(*
SPDX-FileCopyrightText: © 2026 Oleksandr Tiutyk <trofimich@gmail.com>
SPDX-License-Identifier: MIT
License: https://opensource.org/license/mit
*)

(*!
<summary>Creates a filesystem directory through cyclic task execution.</summary>
<description>
Configure DirectoryPath, PathType, AmsNetId and Timeout before Start and keep them unchanged until STOPPED.
The path must be nonblank and pass PathHelper's limited lexical filter; native services determine whether the
requested operation is supported. This task does not perform an existence precheck or suppress native errors.
Invalid configuration and native errors use the base Task failure and cleanup path. Cancellation waits for
submitted I/O without rolling back completed filesystem changes. Reset clears the native request state and
preserves configuration. Use one owner task per instance.
</description>
*)

{attribute 'no_explicit_call' := 'do not call this function block directly'}
FUNCTION_BLOCK CreateDirectory EXTENDS TOF_Tasks.Task IMPLEMENTS IFileSystemTask
VAR_STAT
	//! <summary>Static type metadata available before the base task initializes its default name.</summary>
	{attribute 'hide'}
	_ClassName : STRING := __POUNAME();
END_VAR
VAR
    _CreateDirectory : Tc2_System.FB_CreateDir;
END_VAR

(*!
<summary>Selects the ADS target for the native filesystem operation.</summary>
<description>
Configure before Start and keep unchanged until STOPPED; the setter stores configuration without submitting
I/O.
</description>
*)
{attribute 'monitoring' := 'call'}
PROPERTY AmsNetId : Tc2_System.T_AmsNetID
GET
AmsNetId := _CreateDirectory.sNetId;
END_GET
SET
_CreateDirectory.sNetId := AmsNetId;
END_SET
END_PROPERTY

(*!
<summary>Provides the concrete type name used in diagnostics.</summary>
<description>
Returns borrowed read-only metadata; keep the instance alive and do not modify the referenced string.
Initialized static storage is ready during base Task.FB_init; this getter has no side effects or exceptions.
</description>
*)
{attribute 'monitoring' := 'call'}
PROPERTY ClassName : REFERENCE TO STRING
GET
ClassName REF= _ClassName;
END_GET
END_PROPERTY

{attribute 'monitoring' := 'call'}
(*!
<summary>Provides the copied path for the next directory operation.</summary>
<description>
Set before Start and keep unchanged until STOPPED. Checked by PathHelper before submission, then interpreted
by the native service using PathType. Assignment does not perform I/O; Reset preserves it.
</description>
*)
PROPERTY DirectoryPath : Tc2_System.T_MaxString
GET
DirectoryPath := _CreateDirectory.sPathName;
END_GET
SET
_CreateDirectory.sPathName := DirectoryPath;
END_SET
END_PROPERTY

(*!
<summary>Provides the library namespace used in diagnostics.</summary>
<description>Returns borrowed read-only namespace storage; do not modify the referenced string.</description>
*)
{attribute 'monitoring' := 'call'}
PROPERTY NamespaceName : REFERENCE TO STRING
GET
NamespaceName REF= CurrentNamespace.Name;
END_GET
END_PROPERTY

(*!
<summary>Resets the native request edge after the task has stopped.</summary>
<description>
Preserves configured inputs and does not undo completed filesystem effects. Pending I/O must finish during
stopping before this hook runs.
</description>
*)
METHOD PROTECTED OnReset
_CreateDirectory(bExecute := FALSE);
END_METHOD

(*!
<summary>Validates the configured path and advances the native directory-create request.</summary>
<description>
Computed diagnostic strings are held in local buffers for the duration of the receiving call without dynamic
string-builder allocations.
</description>
*)
METHOD PROTECTED OnRunning
VAR_OUTPUT
	processingState : TOF_Tasks.TASK_PROCESSING_STATE;
END_VAR
VAR_IN_OUT
	stopReasonMessage : TOF_Core.ERROR_MESSAGE;
END_VAR
VAR	
	pathErrorMessage : WSTRING(255);
	formattedExceptionMessage : TOF_Core.ERROR_MESSAGE;
END_VAR
IF NOT _CreateDirectory.bExecute THEN 
	IF TOF_Core.Strings.IsNullOrWhiteSpace(stringToCheck := _CreateDirectory.sPathName) THEN
		TOF_Core.Exceptions.ThrowDataMemberNotSpecified(
			sourceNamespaceName := NamespaceName,
			sourceClassName := ClassName,
			sourcePOUName := __POUNAME(),
			sourcePosition := __POSITION(),
			dataMemberName := 'DirectoryPath'
		);		
	END_IF
	
	IF NOT PathHelper.IsValidDirectoryPath(directoryPath := _CreateDirectory.sPathName, errorMessage => pathErrorMessage) THEN
		FileSystemExceptions.ThrowInvalidPath(
			sourceNamespaceName := NamespaceName,
			sourceClassName := ClassName,
			sourcePOUName := __POUNAME(),
			sourcePosition := __POSITION(),
			path := _CreateDirectory.sPathName,
			errorMessage := pathErrorMessage
		);
	END_IF
END_IF

_CreateDirectory(bExecute := TRUE);

IF _CreateDirectory.bError THEN
	TOF_Core.WideStrings.Append255(
		formattedExceptionMessage,
		"Error while creating directory '",
		TO_WSTRING(_CreateDirectory.sPathName),
		"'");

	FileSystemExceptions.ThrowFileSystem(
		sourceNamespaceName := NamespaceName,
		sourceClassName := ClassName,
		sourcePOUName := __POUNAME(),
		sourcePosition := __POSITION(),
		message := formattedExceptionMessage,
		errorCode := _CreateDirectory.nErrId
	);
ELSIF NOT _CreateDirectory.bBusy THEN
	processingState := TOF_Tasks.TASK_PROCESSING_STATE.DONE;
END_IF
END_METHOD

(*!
<summary>Waits for an already submitted operation before task termination.</summary>
<description>
Runs for every stop reason. Advances the pending FB with bExecute=FALSE without issuing another request.
Completion does not roll back side effects. Keep configuration and borrowed buffers valid until STOPPED.
</description>
<param name="readyToRelease">TRUE when the underlying FB is no longer busy.</param>
*)
METHOD PROTECTED OnStopping
VAR_OUTPUT
	readyToRelease : BOOL;
END_VAR
IF _CreateDirectory.bBusy THEN
	_CreateDirectory(bExecute := FALSE);
END_IF

readyToRelease := NOT _CreateDirectory.bBusy;
END_METHOD

(*!
<summary>Selects the native path context for the filesystem request.</summary>
<description>
Configure before Start and keep unchanged until STOPPED. It is passed to the native operation, not used as a
path-validity result. Reset preserves it.
</description>
*)
{attribute 'monitoring' := 'call'}
PROPERTY PathType : Tc2_System.E_OpenPath
GET
PathType := _CreateDirectory.ePath;
END_GET
SET
_CreateDirectory.ePath := PathType;
END_SET
END_PROPERTY

(*!
<summary>Reports the size of this concrete instance in bytes.</summary>
*)
{attribute 'monitoring' := 'call'}
PROPERTY SelfSize : ULINT
GET
SelfSize := XSIZEOF(THIS^);
END_GET
END_PROPERTY

(*!
<summary>Configures the timeout passed to native operation requests.</summary>
<description>
Set before Start and keep unchanged until STOPPED. Reset preserves this value. It is not an overall task
deadline or a guarantee of resource release after a timeout.
</description>
*)
{attribute 'monitoring' := 'call'}
PROPERTY Timeout : TIME
GET
Timeout := _CreateDirectory.tTimeout;
END_GET
SET
_CreateDirectory.tTimeout := Timeout;
END_SET
END_PROPERTY

END_FUNCTION_BLOCK

(* stored: Version 1.1.0.1
   POU CreateDirectory: Id {7b0b8920-cd1b-44d1-9ca2-1004e427656c}, SpecialFunc None
   Folder Inputs: Id {cd46d3f1-05ad-4d2a-bb18-250033ee445c}
   Folder Members to override: Id {740079d8-792c-4051-b807-b10023f9c7a1}
   Property AmsNetId: Id {ed338df4-10dc-451a-b64d-a000a295e7f0}
   Get Get: Id {94b5c541-fb9b-4788-a387-16d6d7a06a3f}
   Set Set: Id {477e135b-e114-4f7b-ae5e-413843dd690f}
   Property ClassName: Id {68947efb-286a-42af-a556-a0bbd5d3027a}
   Get Get: Id {40a07058-94c4-4be0-ab88-a373f33d3011}
   Property DirectoryPath: Id {7d34ff6b-66c9-43e2-9ce1-01d401372e05}
   Get Get: Id {bfb35ddc-0143-4123-989c-469790325d20}
   Set Set: Id {f1f98b86-e1b0-48a8-a264-70f11718c110}
   Property NamespaceName: Id {ea279b18-2495-419a-af6e-f1db1538b308}
   Get Get: Id {affba913-0ba6-4588-83ed-6a9649f3e1dc}
   Method OnReset: Id {8a28ceca-ec54-49f2-97aa-c7a5fc415861}
   Method OnRunning: Id {6bd810fa-872b-4e47-b2bc-32ff3c16f403}
   Method OnStopping: Id {41f71629-0447-4447-a2fb-74c1ee110012}
   Property PathType: Id {813cddba-24ae-417e-a32e-8078530fc9b5}
   Get Get: Id {26543d70-59ee-403c-af69-d4faa3e2e712}
   Set Set: Id {fc38db83-a1b0-4341-9146-45fe2533fa6e}
   Property SelfSize: Id {ff29508a-b927-484d-8776-c7a1fd61b57a}
   Get Get: Id {9fd144e1-4541-4668-9bfe-274b7a79cf1d}
   Property Timeout: Id {78fb4594-c887-4181-a8a6-4363e1f0945e}
   Get Get: Id {8affc407-c0f2-46cc-acef-d2a177ecaf4b}
   Set Set: Id {0f89e125-a68f-47d7-ab94-803cd70c6f9c} *)
